% RSLogix 500 project P3_ABIOLA_A_V5.RSS, saved by version 8.30.00.16 %
PROJECT "UNTITLED"    % processor: Bul.1763 MicroLogix 1100 Series B %

PROGRAM FILES
  LAD 2   2 rungs
  LAD 3 "PSEUDO IO"  11 rungs  % Contains all the assigned memery address used  %

DATA FILES
  O0 OUTPUT  4 elements
  I1 INPUT  6 elements
  S2 STATUS  66 elements
  B3 BINARY  1 elements
  T4 TIMER  1 elements
  C5 COUNTER  1 elements
  R6 CONTROL  1 elements
  N7 INTEGER  6 elements
  F8 FLOAT  1 elements
  ST9 STRFRBCSCN  5 elements  % Writes string from bar code scanner to PLC %
  ST10 STRING  10 elements

LADDER 2
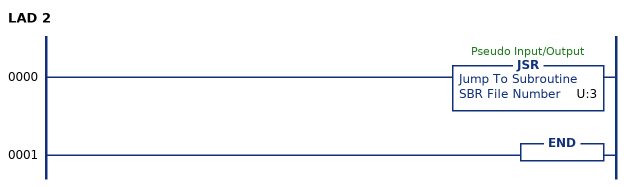
% Rung: 0 %
SOR JSR U:3 EOR
%   U:3  "Pseudo Input/Output" %
% Rung: 1 %
SOR END EOR

LADDER 3 "PSEUDO IO"    % Contains all the assigned memery address used  %
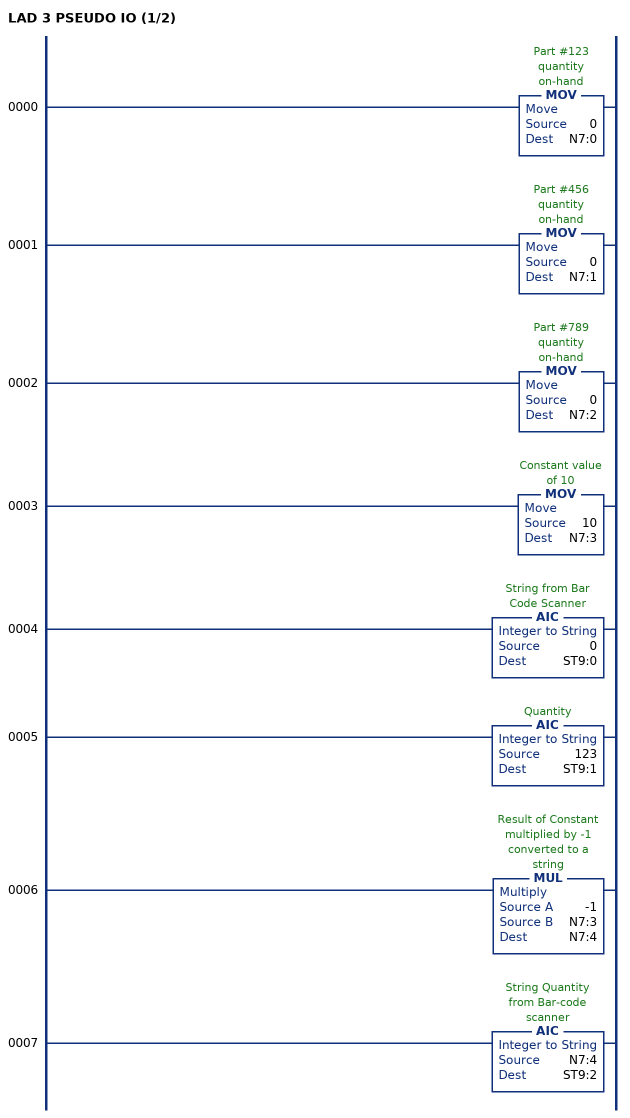
% Rung: 0 %
SOR MOV 0 N7:0 EOR
%   N7:0  "Part #123 quantity on-hand" %
% Rung: 1 %
SOR MOV 0 N7:1 EOR
%   N7:1  "Part #456 quantity on-hand" %
% Rung: 2 %
SOR MOV 0 N7:2 EOR
%   N7:2  "Part #789 quantity on-hand" %
% Rung: 3 %
SOR MOV 10 N7:3 EOR
%   N7:3  "Constant value of 10" %
% Rung: 4 %
SOR AIC 0 ST9:0 EOR
%   ST9:0  "String from Bar Code Scanner" %
% Rung: 5 %
SOR AIC 123 ST9:1 EOR
%   ST9:1  "Quantity" %
% Rung: 6 %
SOR MUL -1 N7:3 N7:4 EOR
%   N7:3  "Constant value of 10" %
%   N7:4  "Result of Constant multiplied by -1 converted to a string" %
% Rung: 7 %
SOR AIC N7:4 ST9:2 EOR
%   N7:4  "Result of Constant multiplied by -1 converted to a string" %
%   ST9:2  "String Quantity from Bar-code scanner" %

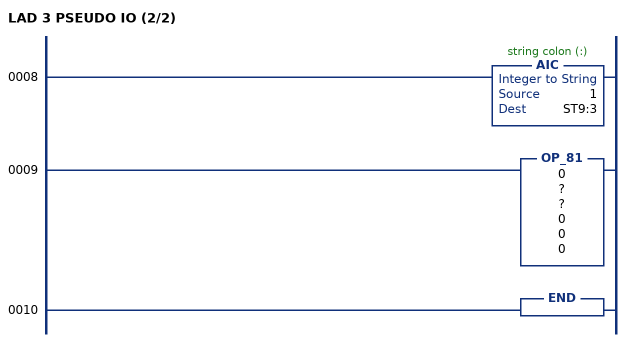
% Rung: 8 %
SOR AIC 1 ST9:3 EOR
%   ST9:3  "string colon (:)" %
% Rung: 9 %  % edit flag set %
SOR OP_81 0 ? ? 0 0 0 EOR
% Rung: 10 %
SOR END EOR

OTHER DOCUMENTED ADDRESSES
  N7:5  "String colon (:) converted to integer"
  ST9:2.0  "Result of Constant Multiplication with -1"
  ST9:4  "Concatination of colon (:) with direction from BCS"
  ST10:1.0  "String len"
